FUNCTION_BLOCK F_PERCENT_TO_FRACTION (* Prozent (REAL 0.0-100.0, z.B. von OPC-UA-Subscribe) in Anteil (REAL 0.0-1.0, fuer F_PWM_PERCENT_TO_RAW.IN) umrechnen und begrenzen *)
  (* Standard: 61499-2; Description: Copyright (c) 2026 Meisterschulen am Ostbahnhof This program and the accompanying materials are made available under the terms of the Eclipse Public License 2.0 which is available at https://www.eclipse.org/legal/epl-2.0/ SPDX-License-Identifier: EPL-2.0 *)
  (* Version 1.0, 2026-08-28, Franz Höpfinger, Meisterschulen am Ostbahnhof, initial API and implementation and/or initial documentation *)
  PACKAGE logiBUS::signalprocessing::fieldbus;
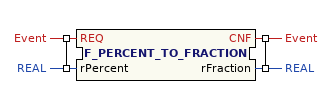
  EVENT_INPUT
    REQ WITH rPercent; (* Umrechnung anfordern *)
  END_EVENT
  EVENT_OUTPUT
    CNF WITH rFraction; (* Umrechnung abgeschlossen *)
  END_EVENT
  VAR_INPUT
    rPercent : REAL; (* Prozentwert, wird auf 0.0-100.0 begrenzt *)
  END_VAR
  VAR_OUTPUT
    rFraction : REAL; (* Anteil 0.0-1.0 *)
  END_VAR
  EC_STATES
    REQ : REQ -> CNF;
  END_STATES
  ALGORITHM REQ IN ST: (* 100.0 % entspricht 1.0, aussenliegende Werte werden geklemmt *)
IF rPercent <= 0.0 THEN
	rFraction := 0.0;
ELSIF rPercent >= 100.0 THEN
	rFraction := 1.0;
ELSE
	rFraction := rPercent / 100.0;
END_IF;
  END_ALGORITHM
END_FUNCTION_BLOCK
